# EPICS substitutions: iocBoot/iocNSLS2I_EM/DACs.substitutions
file "$(QUADEM)/db/NSLS2_DAC.template"
{
pattern
{P,               R,     N, PORT,     EGUL,   DRVL,  LOPR,  EGUF,  DRVH,   HOPR, PREC,  LINR}
{quadEMTest:, NSLS2I_EM:, 0, NSLS2I_EM,  -10,   -10,   -10,    10,   10.,    10.,  4,     LINEAR}
{quadEMTest:, NSLS2I_EM:, 1, NSLS2I_EM,  -10,   -10,   -10,    10,   10.,    10.,  4,     LINEAR}
{quadEMTest:, NSLS2I_EM:, 2, NSLS2I_EM,  -10,   -10,   -10,    10,   10.,    10.,  4,     LINEAR}
{quadEMTest:, NSLS2I_EM:, 3, NSLS2I_EM,  -10,   -10,   -10,    10,   10.,    10.,  4,     LINEAR}
}
